FUNCTION_BLOCK FB_SITP_SygnalizacjaStanu_Suspended EXTENDS FB_SITP_SygnalizacjaStanu
VAR
END_VAR

METHOD PUBLIC UstawPrace
VAR_INPUT
END_VAR

THIS^.refarrLampki [E_SITP_LampkiSygnalizacyjne.WiezaCzerwona].Wlacz2		(bSwiec := FALSE, 	bMigaj := FALSE,	 tWlaczony := T#0MS,	 tWylaczony := T#0MS);(*			Czerwona		*)
THIS^.refarrLampki [E_SITP_LampkiSygnalizacyjne.WiezaZolta].Wlacz2			(bSwiec := FALSE, 	bMigaj := TRUE,		 tWlaczony := T#400MS,	 tWylaczony := T#400MS);(*			Zółta			*)
THIS^.refarrLampki [E_SITP_LampkiSygnalizacyjne.WiezaZielona].Wlacz2		(bSwiec := TRUE, 	bMigaj := FALSE,	 tWlaczony := T#0MS,	 tWylaczony := T#0MS);(*			Zielona			*)
THIS^.refarrLampki [E_SITP_LampkiSygnalizacyjne.WiezaBiala].Wlacz2			(bSwiec := FALSE, 	bMigaj := FALSE,	 tWlaczony := T#0MS,	 tWylaczony := T#0MS);(*			Niebieska		*)
THIS^.refarrLampki [E_SITP_LampkiSygnalizacyjne.WiezaNiebieska].Wlacz2		(bSwiec := FALSE, 	bMigaj := FALSE,	 tWlaczony := T#0MS,	 tWylaczony := T#0MS);(*			Biała			*)



THIS^.refarrLampki [E_SITP_LampkiSygnalizacyjne.PrzyciskStart].Wlacz2		(bSwiec := TRUE, 	bMigaj := FALSE,	 tWlaczony := T#0MS,	 tWylaczony := T#0MS);(*	Lampka przycisku Start    	*)
THIS^.refarrLampki [E_SITP_LampkiSygnalizacyjne.PrzyciskStop].Wlacz2		(bSwiec := FALSE, 	bMigaj := FALSE,	 tWlaczony := T#0MS,	 tWylaczony := T#0MS);(*	Lampka przycisku Stop     	*)
THIS^.refarrLampki [E_SITP_LampkiSygnalizacyjne.PrzyciskHold].Wlacz2		(bSwiec := FALSE, 	bMigaj := FALSE,	 tWlaczony := T#0MS,	 tWylaczony := T#0MS);(*	Lampka przycisku Hold     	*)
THIS^.refarrLampki [E_SITP_LampkiSygnalizacyjne.PrzyciskUnhold].Wlacz2		(bSwiec := FALSE, 	bMigaj := FALSE,	 tWlaczony := T#0MS,	 tWylaczony := T#0MS);(*	Lampka przycisku Unhold   	*)
THIS^.refarrLampki [E_SITP_LampkiSygnalizacyjne.PrzyciskSuspend].Wlacz2		(bSwiec := FALSE, 	bMigaj := FALSE,	 tWlaczony := T#0MS,	 tWylaczony := T#0MS);(*	Lampka przycisku Suspend  	*)
THIS^.refarrLampki [E_SITP_LampkiSygnalizacyjne.PrzyciskUnsuspend].Wlacz2	(bSwiec := FALSE, 	bMigaj := FALSE,	 tWlaczony := T#0MS,	 tWylaczony := T#0MS);(*	Lampka przycisku Unsuspend	*)
THIS^.refarrLampki [E_SITP_LampkiSygnalizacyjne.PrzyciskAbort].Wlacz2		(bSwiec := FALSE, 	bMigaj := FALSE,	 tWlaczony := T#0MS,	 tWylaczony := T#0MS);(*	Lampka przycisku Abort    	*)
THIS^.refarrLampki [E_SITP_LampkiSygnalizacyjne.PrzyciskClear].Wlacz2		(bSwiec := FALSE, 	bMigaj := FALSE,	 tWlaczony := T#0MS,	 tWylaczony := T#0MS);(*	Lampka przycisku Clear    	*)
THIS^.refarrLampki [E_SITP_LampkiSygnalizacyjne.PrzyciskComplete].Wlacz2	(bSwiec := FALSE, 	bMigaj := FALSE,	 tWlaczony := T#0MS,	 tWylaczony := T#0MS);(*	Lampka przycisku Complete	*)
END_METHOD

END_FUNCTION_BLOCK

(* stored: Version 1.1.0.1
   POU FB_SITP_SygnalizacjaStanu_Suspended: Id {d35009ca-57d3-051e-1845-0ad96d598693}, SpecialFunc None
   Method UstawPrace: Id {1c9a989d-1324-0479-0eea-ab00da190243} *)
